// TwinCAT 3 PLC project PLC
// ProgramVersion: 3.1.4026.14
// libraries:
//   Tc2_Standard, * (Beckhoff Automation GmbH)
//   Tc2_System, * (Beckhoff Automation GmbH)
//   Tc2_Utilities, * (Beckhoff Automation GmbH)
// project tree:
//   / PlcTask.TcTTO
//   POUs/ FB_StateMachine.TcPOU, MAIN.TcPOU
// real-time tasks:
//   TASK PlcTask: cycle T#10ms, priority 20, ADS port 350

CONFIGURATION PLC
    RESOURCE PLC ON TwinCAT3
        TASK PlcTask(INTERVAL := T#10ms, PRIORITY := 20);
        PROGRAM MAIN WITH PlcTask : MAIN;
    END_RESOURCE
END_CONFIGURATION

// ---- POUs/MAIN.TcPOU
PROGRAM MAIN
VAR
	StateMachine : FB_StateMachine;
	hr			 : HRESULT;

	//I_StateMachine 	
	Start : BOOL;
	Stop  : BOOL;
	State : INT;

	//ITComObject
	SetTcCOMState	   : BOOL;
	NewState		   : TCOM_STATE := TCOM_STATE.TCOM_STATE_PREOP;
	GetTcComState	   : BOOL;
	ActState		   : TCOM_STATE;
	GetParam, SetParam : BOOL;
	SizeOfState		   : UDINT;
	PointerToState	   : POINTER TO INT;
	Param_State		   : INT;

	//ITCADI	
	PointerToInputs	 : POINTER TO INT;
	PointerToOutputs : POINTER TO INT;
	GetIn1, SetIn1	 : BOOL;
	In1				 : INT;
	GetOut1, SetOut1 : BOOL;
	Out1			 : INT;
END_VAR

//I_StateMachine 
IF StateMachine.ip_StateMachine <> 0 THEN
	IF Start THEN
		StateMachine.ip_StateMachine.M_Start();
		Start := FALSE;
	END_IF

	IF Stop THEN
		StateMachine.ip_StateMachine.M_Stop();
		Stop := FALSE;
	END_IF

	StateMachine.ip_StateMachine.M_GetState(State);
END_IF

//ITComObject
IF StateMachine.ip_ComObject <> 0 THEN
	IF SetTcCOMState THEN
		SetTcCOMState := FALSE;
		hr			  := StateMachine.ip_ComObject.TcSetObjState(state := NewState, ipSrv := TwinCAT_SystemInfoVarList._AppInfo.TComSrvPtr, pInitData := 0);
	END_IF

	IF GetTcComState THEN
		GetTcComState := FALSE;
		hr			  := StateMachine.ip_ComObject.TcGetObjState(ADR(ActState));
	END_IF

	IF GetParam OR SetParam THEN
		SizeOfState	   := SIZEOF(Param_State);
		PointerToState := ADR(Param_State);
	END_IF

	IF GetParam THEN
		GetParam := FALSE;
		hr		 := StateMachine.ip_ComObject.TcGetObjPara(pid	 := 16#1,
														   nData := SizeOfState,
														   pData := PointerToState,
														   0);
	END_IF

	IF SetParam THEN
		SetParam := FALSE;
		hr		 := StateMachine.ip_ComObject.TcSetObjPara(pid	 := 16#1,
														   nData := SizeOfState,
														   pData := PointerToState,
														   0);
	END_IF
END_IF

//ITCADI
IF StateMachine.ip_DataArea <> 0 THEN
	IF GetIn1 THEN
		GetIn1 := FALSE;
		hr	   := StateMachine.ip_DataArea.GetImagePtr(size	  := SIZEOF(In1),
													   offs	  := 0,
													   adi_x  := 1,
													   ppData := ADR(PointerToInputs));

		IF hr = S_OK THEN
			MEMCPY(destAddr := ADR(In1), srcAddr := PointerToInputs, n := SIZEOF(In1));
			hr := StateMachine.ip_DataArea.ReleaseImagePtr(PointerToInputs);
		END_IF
	END_IF

	IF SetIn1 THEN
		SetIn1 := FALSE;
		hr	   := StateMachine.ip_DataArea.GetImagePtr(size	  := SIZEOF(In1),
													   offs	  := 0,
													   adi_x  := 1,
													   ppData := ADR(PointerToInputs));

		IF hr = S_OK THEN
			MEMCPY(destAddr := PointerToInputs, srcAddr := ADR(In1), n := SIZEOF(In1));
			hr := StateMachine.ip_DataArea.ReleaseImagePtr(PointerToInputs);
		END_IF
	END_IF

	IF GetOut1 THEN
		GetOut1 := FALSE;
		hr		:= StateMachine.ip_DataArea.GetImagePtr(size   := SIZEOF(Out1),
														offs   := 0,
														adi_x  := 2,
														ppData := ADR(PointerToOutputs));

		IF hr = S_OK THEN
			MEMCPY(destAddr := ADR(Out1), srcAddr := PointerToOutputs, n := SIZEOF(Out1));
			hr := StateMachine.ip_DataArea.ReleaseImagePtr(PointerToOutputs);
		END_IF
	END_IF

	IF SetOut1 THEN
		SetOut1 := FALSE;
		hr		:= StateMachine.ip_DataArea.GetImagePtr(size   := SIZEOF(Out1),
														offs   := 0,
														adi_x  := 2,
														ppData := ADR(PointerToOutputs));

		IF hr = S_OK THEN
			MEMCPY(destAddr := PointerToOutputs, srcAddr := ADR(Out1), n := SIZEOF(Out1));
			hr := StateMachine.ip_DataArea.ReleaseImagePtr(PointerToOutputs);
		END_IF
	END_IF
END_IF

END_PROGRAM

// ---- POUs/FB_StateMachine.TcPOU
FUNCTION_BLOCK FB_StateMachine
VAR_INPUT
	ip_StateMachine : I_StateMachine;
	ip_ComObject	: ITComObject;
	ip_DataArea		: ITCADI;
END_VAR

VAR
	{attribute 'TcInitSymbol'}
	oid				 : OTCID;
	hrStateMachine	 : HRESULT;
	iid_StateMachine : IID := TC_GLOBAL_IID_LIST.IID_I_StateMachine;
	hrGetInstance	 : HRESULT;
	iid_TcCOMObject	 : IID := TC_GLOBAL_IID_LIST.IID_ITComObject;
	hrITcADI		 : HRESULT;
	iid_ITcADI		 : IID := TC_GLOBAL_IID_LIST.IID_ITcADI;
END_VAR

//FB_Exit must be implemented explicitly. If there is an implementation, then the

//method is called before the controller removes the code of the function block instance

//(implicit call). The return value is not evaluated.
METHOD FB_Exit : BOOL
VAR_INPUT
	bInCopyCode : BOOL; // TRUE: the exit method is called in order to leave the instance which will be copied afterwards (online change).  
END_VAR
IF NOT bInCopyCode THEN
	FW_SafeRelease(ADR(ip_StateMachine));
	FW_SafeRelease(ADR(ip_ComObject));
	FW_SafeRelease(ADR(ip_DataArea));
END_IF
END_METHOD

//FB_Init is always available implicitly and it is used primarily for initialization.

//The return value is not evaluated. For a specific influence, you can also declare the

//methods explicitly and provide additional code there with the standard initialization

//code. You can evaluate the return value.
METHOD FB_Init : BOOL
VAR_INPUT
	bInitRetains : BOOL; // TRUE: the retain variables are initialized (reset warm / reset cold)
	bInCopyCode	 : BOOL; // TRUE: the instance will be copied to the copy code afterward (online change)  
END_VAR
IF NOT bInCopyCode THEN
	hrStateMachine := FW_ObjMgr_GetObjectInstance(oid := oid, iid := iid_StateMachine, ADR(ip_StateMachine));
	hrStateMachine := FW_ObjMgr_GetObjectInstance(oid := oid, iid := iid_TcCOMObject, ADR(ip_ComObject));
	hrITcADI	   := FW_ObjMgr_GetObjectInstance(oid := oid, iid := iid_ITcADI, ADR(ip_DataArea));
END_IF
END_METHOD

END_FUNCTION_BLOCK
